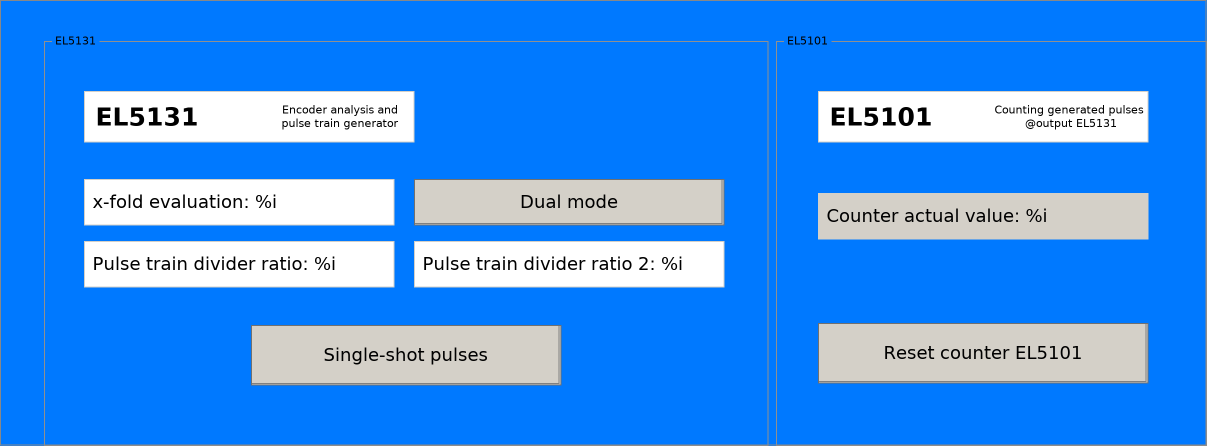
VISUALIZATION MAINVISU  // 1207x446
    GroupBox (44,33 724x413), "EL5131"
        Textfield (370,208 310x46), "Pulse train divider ratio 2: %i", text variable: MAINEL5131.iDivRatio2, invisible if: not MAINEL5131.bDualMode
            OnMouseClick: write the text variable via VisuDialogs.Numpad, min 2, max 20
        Button (370,146 310x46), "Dual mode"
            toggle MAINEL5131.bDualMode
        Textfield (40,146 310x46), "x-fold evaluation: %i", text variable: MAINEL5131.iEvalMode
            OnMouseClick: write the text variable via VisuDialogs.Numpad, min 1, max 4
        Button (207,292 310x60), "Single-shot pulses"
            toggle MAINEL5131.bSingleShot
    Textfield (84,91 330x51), "EL5131"
    Textfield (84,241 310x46), "Pulse train divider ratio: %i", text variable: MAINEL5131.iDivRatio
        OnMouseClick: write the text variable via VisuDialogs.Numpad, min 2, max 20
    Label (262,95 156x43), "Encoder analysis and pulse train generator"
    GroupBox (776,33 431x413), "EL5101"
    Textfield (818,91 330x51), "EL5101"
    Textfield (818,193 330x46), "Counter actual value: %i", text variable: MAIN.iCounterValueDoubleCheckEL5101
    Button (818,323 330x60), "Reset counter EL5101"
        tap MAIN.bResetEL5101
    Label (993,95 156x43), "Counting generated pulses @output EL5131"
END_VISUALIZATION

(* stored: Version 1.1.0.1, ProductVersion 3.1.4024.11
   Visu MAINVISU: Id {796d719c-4d7c-4b4d-a0eb-a62729f1c65d} *)
